TYPE StepperPOSStatus :
STRUCT
	Busy : BOOL;
	InTarget : BOOL;
	Warning : BOOL;
	Error : BOOL;
	Calibrated : BOOL;
	Accelerate : BOOL;
	Decelerate : BOOL;
	ReadyToExecute : BOOL;
	ActualPosition : UDINT;
	ActualVelocity : INT;
	ActualDriveTime : UDINT;
END_STRUCT
END_TYPE

(* stored: Version 1.1.0.1, ProductVersion 3.1.4024.11
   DUT StepperPOSStatus: Id {1a121297-b503-41ac-a804-890c986b25bb} *)
